// TIA Portal V17 export
// export: Created 2024-09-03T21:54:50.1601534Z, ExportSetting WithDefaults, DisplayName Totally Integrated Automation Portal, DisplayVersion V17 Update 7, DisplayName TIA Portal Openness, DisplayVersion V17 Update 7, DisplayName TIA Portal Version Control Interface, DisplayVersion V17, DisplayName SINAMICS Startdrive Advanced, DisplayVersion V17 SP2, DisplayName SINAMICS Startdrive G110M, G120, G120C, G120D, G120P, G115D, DisplayVersion V17 SP2, DisplayName SINAMICS Startdrive G130, G150, S120, S150, SINAMICS MV, S210, DisplayVersion V17 SP2, DisplayName STEP 7 Professional, DisplayVersion V17 Update 7, DisplayName STEP 7 Safety, DisplayVersion V17 Update 6, DisplayName WinCC Advanced / Unified PC, DisplayVersion V17 Update 7
DATA_BLOCK "IODiagnostic_DB"   // DB18
VERSION : 0.1
// stored: AutoNumber true, DBAccessibleFromOPCUA true, DBAccessibleFromWebserver true, InstanceOfName IODiagnostic, InstanceOfType FB
"IODiagnostic"
   // VAR
   //    DeviceNumber : Int := 0;
   //    DeviceNumberOld : Int := 0;
   //    InputAdress : Int := 0;
   //    OutputAdress : Int := 0;
   //    InputImage : Array[1.."IOImageSize"] of Byte;
   //    OutputImage : Array[1.."IOImageSize"] of Byte;
   //    InputAdresses : Array[1.."IOImageSize"] of Int;
   //    OutputAdresses : Array[1.."IOImageSize"] of Int;
   //    SingleAdressInput : Int := 0;
   //    SingleAdressOutput : Int := 0;
   //    SingleInput : Byte := 16#06;
   //    SingleOutput : Byte := 16#00;
   //    res : Byte := 16#00;
   // END_VAR
BEGIN
   InputImage[1] := 16#06;
   InputImage[2] := 16#C0;
   InputImage[3] := 16#84;
   InputImage[4] := 16#00;
   InputImage[5] := 16#C4;
   InputImage[6] := 16#42;
   InputImage[7..14] := 16#00;
   InputImage[15] := 16#0F;
   InputImage[16..20] := 16#00;
   OutputImage[1] := 16#00;
   OutputImage[2] := 16#04;
   OutputImage[3] := 16#20;
   OutputImage[4..14] := 16#00;
   OutputImage[15] := 16#0F;
   OutputImage[16] := 16#A0;
   OutputImage[17] := 16#48;
   OutputImage[18] := 16#EE;
   OutputImage[19] := 16#14;
   OutputImage[20] := 16#00;
   InputAdresses[1] := 0;
   InputAdresses[2] := 1;
   InputAdresses[3] := 2;
   InputAdresses[4] := 3;
   InputAdresses[5] := 4;
   InputAdresses[6] := 5;
   InputAdresses[7] := 6;
   InputAdresses[8] := 7;
   InputAdresses[9] := 8;
   InputAdresses[10] := 9;
   InputAdresses[11] := 10;
   InputAdresses[12] := 11;
   InputAdresses[13] := 12;
   InputAdresses[14] := 13;
   InputAdresses[15] := 14;
   InputAdresses[16] := 15;
   InputAdresses[17] := 16;
   InputAdresses[18] := 17;
   InputAdresses[19] := 18;
   InputAdresses[20] := 19;
   OutputAdresses[1] := 0;
   OutputAdresses[2] := 1;
   OutputAdresses[3] := 2;
   OutputAdresses[4] := 3;
   OutputAdresses[5] := 4;
   OutputAdresses[6] := 5;
   OutputAdresses[7] := 6;
   OutputAdresses[8] := 7;
   OutputAdresses[9] := 8;
   OutputAdresses[10] := 9;
   OutputAdresses[11] := 10;
   OutputAdresses[12] := 11;
   OutputAdresses[13] := 12;
   OutputAdresses[14] := 13;
   OutputAdresses[15] := 14;
   OutputAdresses[16] := 15;
   OutputAdresses[17] := 16;
   OutputAdresses[18] := 17;
   OutputAdresses[19] := 18;
   OutputAdresses[20] := 19;
END_DATA_BLOCK
